TYPE "DeltaPressure"
VERSION : 0.1
   STRUCT
      Val : "Val";
      Limits : "Limits";
   END_STRUCT;

END_TYPE

